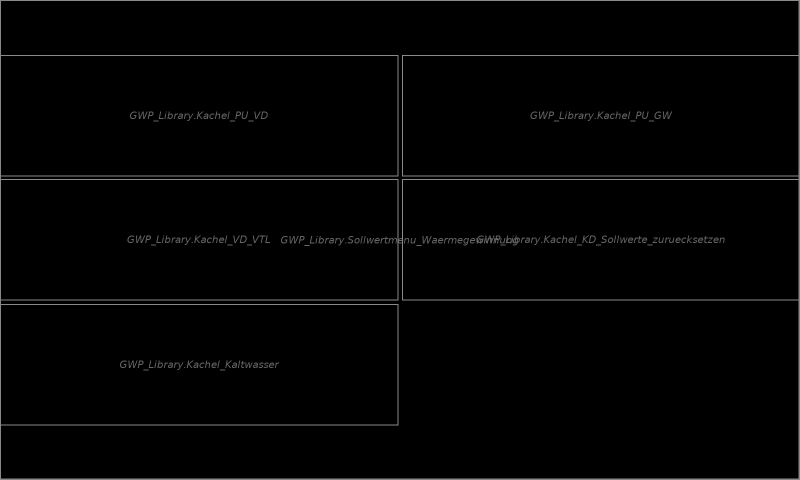
VISUALIZATION Sollwertmenu_Waermegewinnung  // 800x480
    Frame (0,0 800x480)
        shows GWP_Library.Sollwertmenu_Waermegewinnung(FB_KWP_SP_AC_NC := Main.KWP_SP_AC_NC_0, FB_Kreis_3KO := Main.Kreis_3KO_0, FB_Init_1 := Main.Init_0)
    Frame (0,55 398x121)
        shows GWP_Library.Kachel_PU_VD()
        OnMouseClick: change screen: VD_PU_Sollwerte
    Frame (402,55 398x121)
        shows GWP_Library.Kachel_PU_GW()
        OnMouseClick: change screen: VD_GW_Sollwerte
    Frame (0,304 398x121)
        shows GWP_Library.Kachel_Kaltwasser(FB_Kreis_3KO := Main.Kreis_3KO_0)
        OnMouseClick: change screen: Sollwertmenu_KWP
    Frame (402,179 398x121)
        shows GWP_Library.Kachel_KD_Sollwerte_zuruecksetzen()
        OnMouseClick: change screen: VD_Sollwerte_zuruecksetzen
    Frame (0,179 398x121)
        shows GWP_Library.Kachel_VD_VTL()
        OnMouseClick: change screen: VD_VTL_Sollwerte
END_VISUALIZATION

(* stored: Version 1.1.0.1, ProductVersion 3.1.4022.6
   Visu Sollwertmenu_Waermegewinnung: Id {918fecb8-0acf-4d0d-a5ca-af27b60c636a} *)
